// TwinCAT 3 PLC project TcUnit
// Title: TcUnit
// Company: www.tcunit.org
// Author: Jakob Sagatowski and contributors
// ProjectVersion: 1.2.0.0
// Description: TwinCAT unit testing framework. Documentation and examples are available at www.tcunit.org
// ProgramVersion: 3.1.4023.0
// libraries:
//   SysDir, * (System)
//   SysFile, * (System)
//   Tc2_Standard, * (Beckhoff Automation GmbH)
//   Tc2_System, * (Beckhoff Automation GmbH)
//   Tc2_Utilities, * (Beckhoff Automation GmbH)
//   Base Interfaces,newest,System
// project tree:
//   DUTs/ E_AssertionType.TcDUT (not stored), E_XmlError.TcDUT (not stored), ST_AdsLogStringMessage.TcDUT (not stored), ST_AssertResult.TcDUT (not stored), ST_AssertResultInstances.TcDUT (not stored), ST_AssertArrayResult.TcDUT (not stored), ST_AssertArrayResultInstances.TcDUT (not stored), ST_TestCaseResult.TcDUT (not stored), ST_TestSuiteResult.TcDUT (not stored), ST_TestSuiteResults.TcDUT (not stored), U_ExpectedOrActual.TcDUT (not stored)
//   GVLs/ GVL_Param_TcUnit.TcGVL (not stored), GVL_TcUnit.TcGVL (not stored)
//   ITFs/ I_AssertMessageFormatter.TcIO (not stored), I_TestResultLogger.TcIO (not stored), I_TestResults.TcIO (not stored)
//   POUs/ FB_AdsAssertMessageFormatter.TcPOU (not stored), FB_AdsLogStringMessageFifoQueue.TcPOU (not stored), FB_AdsTestResultLogger.TcPOU (not stored), FB_FileControl.TcPOU (not stored), FB_StreamBuffer.TcPOU (not stored), FB_xUnitXmlPublisher.TcPOU (not stored), FB_TestResults.TcPOU (not stored), FB_AdjustAssertFailureMessageToMax253CharLength.TcPOU (not stored), FB_AssertResultStatic.TcPOU (not stored), FB_AssertArrayResultStatic.TcPOU (not stored), FB_TcUnitRunner.TcPOU (not stored), FB_Test.TcPOU (not stored), FB_TestSuite.TcPOU (not stored), FB_XmlControl.TcPOU (not stored)
//   POUs/Functions/ F_AnyToUnionValue.TcPOU (not stored), F_AnyTypeClassToString.TcPOU (not stored), F_AssertionTypeToString.TcPOU (not stored), F_GetTestSuiteNameFromTestInstancePath.TcPOU (not stored), F_IsAnyEqualToUnionValue.TcPOU (not stored), F_RemoveInstancePathAndProjectNameFromTestInstancePath.TcPOU (not stored), IS_TEST_FINISHED.TcPOU (not stored), RUN.TcPOU (not stored), RUN_IN_SEQUENCE.TcPOU (not stored), TCUNIT_ADSLOGSTR.TcPOU (not stored), TEST.TcPOU (not stored), TEST_FINISHED.TcPOU (not stored), TEST_FINISHED_NAMED.TcPOU (not stored), TEST_ORDERED.TcPOU (not stored)
//   POUs/Functions/WRITE_PROTECTED_/ WRITE_PROTECTED_BOOL.TcPOU (not stored), WRITE_PROTECTED_BYTE.TcPOU (not stored), WRITE_PROTECTED_DATE.TcPOU (not stored), WRITE_PROTECTED_DATE_AND_TIME.TcPOU (not stored), WRITE_PROTECTED_DINT.TcPOU (not stored), WRITE_PROTECTED_DWORD.TcPOU (not stored), WRITE_PROTECTED_INT.TcPOU (not stored), WRITE_PROTECTED_LREAL.TcPOU (not stored), WRITE_PROTECTED_REAL.TcPOU (not stored), WRITE_PROTECTED_SINT.TcPOU (not stored), WRITE_PROTECTED_STRING.TcPOU (not stored), WRITE_PROTECTED_WSTRING.TcPOU (not stored), WRITE_PROTECTED_TIME.TcPOU (not stored), WRITE_PROTECTED_TIME_OF_DAY.TcPOU (not stored), WRITE_PROTECTED_UDINT.TcPOU (not stored), WRITE_PROTECTED_UINT.TcPOU (not stored), WRITE_PROTECTED_ULINT.TcPOU (not stored), WRITE_PROTECTED_LWORD.TcPOU (not stored), WRITE_PROTECTED_LINT.TcPOU (not stored), WRITE_PROTECTED_USINT.TcPOU, WRITE_PROTECTED_WORD.TcPOU
//   Version/ Global_Version.TcGVL

// ---- Version/Global_Version.TcGVL
{attribute 'TcGenerated'}
{attribute 'no-analysis'}
{attribute 'linkalways'}
// This function has been automatically generated from the project information.
VAR_GLOBAL CONSTANT
	{attribute 'const_non_replaced'}
	stLibVersion_TcUnit : ST_LibVersion := (iMajor := 1, iMinor := 2, iBuild := 0, iRevision := 0, sVersion := '1.2.0.0');
END_VAR

// ---- POUs/Functions/WRITE_PROTECTED_/WRITE_PROTECTED_USINT.TcPOU
FUNCTION WRITE_PROTECTED_USINT
VAR_INPUT
    Ptr : POINTER TO USINT;
    Value : USINT;
END_VAR

Ptr^ := Value;

END_FUNCTION

// ---- POUs/Functions/WRITE_PROTECTED_/WRITE_PROTECTED_WORD.TcPOU
FUNCTION WRITE_PROTECTED_WORD
VAR_INPUT
    Ptr : POINTER TO WORD;
    Value : WORD;
END_VAR

Ptr^ := Value;

END_FUNCTION
